INTERFACE I_LinkedObject EXTENDS I_Object

PROPERTY ipContext : I_Context
GET
END_GET
END_PROPERTY

PROPERTY ipParent : I_LinkedObject
GET
END_GET
END_PROPERTY

END_INTERFACE

(* stored: Version 1.1.0.1, ProductVersion 3.1.4024.12
   Itf I_LinkedObject: Id {7d3a4e56-9527-01fc-1a73-2082b1d8ceca}
   Property ipContext: Id {d54a9832-a1de-45c3-9205-7c8581f64604}
   Get Get: Id {f2c6904c-7ca9-4293-8141-7b24b0bbbb4d}
   Property ipParent: Id {2c0a360e-cfc4-0237-1414-097f4fc2748c}
   Get Get: Id {d5eab88b-5363-0f33-3e6e-472a6b3fdf68} *)
